// TIA Portal V17 export
// export: Created 2022-04-06T07:28:40.1687276Z, ExportSetting WithDefaults, DisplayName Totally Integrated Automation Portal, DisplayVersion V17, DisplayName TIA Portal Openness, DisplayVersion V17, DisplayName TIA Portal Version Control Interface, DisplayVersion V17, DisplayName TIA Portal Test Suite Advanced, DisplayVersion V17, DisplayName SINAMICS Startdrive Advanced, DisplayVersion V17, DisplayName SINAMICS Startdrive G130, G150, S120, S150, SINAMICS MV, S210, DisplayVersion V17, DisplayName SINAMICS Startdrive G110M, G120, G120C, G120D, G120P, G115D, DisplayVersion V17, DisplayName STEP 7 Professional, DisplayVersion V17, DisplayName STEP 7 Safety, DisplayVersion V17, DisplayName WinCC Advanced / Unified PC, DisplayVersion V17
DATA_BLOCK "Motion_DB"   // DB5
VERSION : 0.1
// stored: AutoNumber true, DBAccessibleFromOPCUA true, DBAccessibleFromWebserver true, InstanceOfName Motion, InstanceOfType FB
"Motion"
   // VAR
   //    MC_POWER_Instance { S7_SetPoint := 'True'} : MC_POWER;
   //    MC_RESET_Instance { S7_SetPoint := 'True'} : MC_RESET;
   //    MC_HOME_Instance { S7_SetPoint := 'True'} : MC_HOME;
   //    MC_MOVEVELOCITY_Instance { S7_SetPoint := 'True'} : MC_MOVEVELOCITY;
   //    MC_HALT_Instance { S7_SetPoint := 'True'} : MC_HALT;
   //    MC_POWER_Instance_1 { S7_SetPoint := 'True'} : MC_POWER;
   //    MC_RESET_Instance_1 { S7_SetPoint := 'True'} : MC_RESET;
   //    MC_HOME_Instance_1 { S7_SetPoint := 'True'} : MC_HOME;
   //    MC_MOVEVELOCITY_Instance_1 { S7_SetPoint := 'True'} : MC_MOVEVELOCITY;
   //    MC_HALT_Instance_1 { S7_SetPoint := 'True'} : MC_HALT;
   //    instMC_MOVEVELOCITY_SlsActive { S7_SetPoint := 'True'} : MC_MOVEVELOCITY;
   //    statSlsPtrig { S7_SetPoint := 'True'} : Bool;
   // END_VAR
BEGIN
END_DATA_BLOCK
